FUNCTION_BLOCK SampleSequence EXTENDS CyclicBase
VAR
	ThisMover : I_XtsMoverAxis;
	LeaveTest: BOOL;
	ArriveTest: BOOL;
	TestMove: BOOL;
	Position: MC_LREAL;
	Velocity: MC_LREAL;
END_VAR

METHOD PUBLIC  Cycle : HRESULT
VAR_INPUT
END_VAR
IF LeaveTest THEN
	MyMover.TriggerMoverLeave();
END_IF

IF ArriveTest THEN
	MyMover.TriggerMoverArrive();
END_IF

IF TestMove THEN
	MyMover.MoveTo(RequiredPosition := Position, MoveVelocity := Velocity);
	TestMove := FALSE;
END_IF
END_METHOD

METHOD FB_init : BOOL
VAR_INPUT
	bInitRetains : BOOL; // if TRUE, the retain variables are initialized (warm start / cold start)
	bInCopyCode : BOOL;  // if TRUE, the instance afterwards gets moved into the copy code (online change)
	XtsRunner : I_ObjectRunner;
END_VAR
XtsRunner.AddComponent(THIS^);
END_METHOD

PROPERTY MyMover : I_XtsMoverAxis
GET
MyMover := ThisMover;
END_GET
SET
ThisMover := MyMover;
END_SET
END_PROPERTY

END_FUNCTION_BLOCK

(* stored: Version 1.1.0.1, ProductVersion 3.1.4024.12
   POU SampleSequence: Id {aeca387d-57da-4277-9b3c-59b22eeb58f8}, SpecialFunc None
   Method Cycle: Id {e67454eb-585e-4a43-aa27-1301f6d081d1}
   Method FB_init: Id {b21bcb06-91a6-46b3-bb9d-ed6a9a698452}
   Property MyMover: Id {c23dd5f6-58df-442d-9989-7b1384c2b3ac}
   Get Get: Id {b9d1641a-aa56-4f84-90c7-004f2597e2ee}
   Set Set: Id {5ca29307-712f-4ddb-a5e2-33d69141bb16} *)
